Omron CX-Programmer project NewProject (CX-Programmer 9.61)

# PLC PLC_Pick: CP1H XA

## Global symbols (name address type ; comment)
0.00 BOOL  ; Start
0.01 BOOL  ; EmitBox
0.02 BOOL  ; EmitBox2
0.03 BOOL  ; Stop
0.04 BOOL  ; Dif1
0.05 BOOL  ; Dif2
0.06 BOOL  ; GrabDet
0.07 BOOL  ; Dif3
0.08 BOOL  ; Dif4
100.00 BOOL  ; M1
100.01 BOOL  ; M2
100.02 BOOL  ; M3
100.03 BOOL  ; M4
100.04 BOOL  ; M4
10.00 BOOL  ; Con6m
10.01 BOOL  ; Con2m1
10.02 BOOL  ; Con2m2
10.03 BOOL  ; BoxEmitter
10.04 BOOL  ; StoperRoll
10.05 BOOL  ; MZ
10.06 BOOL  ; MX
10.07 BOOL  ; Grab
10.08 BOOL  ; StoperBlade
T0000 BOOL  ; Timer1
T0001 BOOL  ; Timer2
T0002 BOOL  ; Timer3

## Program NewProgram1 (cyclic task 0)

### Section Section1

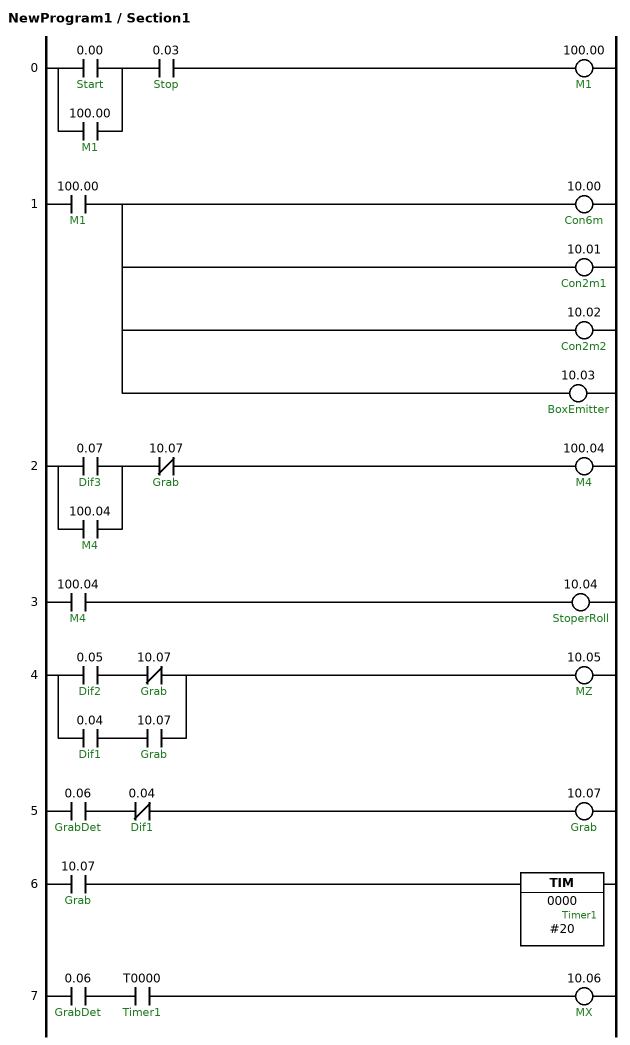
; rung 0
LD 0.00  ; Start
OR 100.00  ; M1
AND 0.03  ; Stop
OUT 100.00  ; M1
; rung 1
LD 100.00  ; M1
OUT 10.00  ; Con6m
OUT 10.01  ; Con2m1
OUT 10.02  ; Con2m2
OUT 10.03  ; BoxEmitter
; rung 2
LD 0.07  ; Dif3
OR 100.04  ; M4
ANDNOT 10.07  ; Grab
OUT 100.04  ; M4
; rung 3
LD 100.04  ; M4
OUT 10.04  ; StoperRoll
; rung 4
LD 0.05  ; Dif2
ANDNOT 10.07  ; Grab
LD 0.04  ; Dif1
AND 10.07  ; Grab
ORLD
OUT 10.05  ; MZ
; rung 5
LD 0.06  ; GrabDet
ANDNOT 0.04  ; Dif1
OUT 10.07  ; Grab
; rung 6
LD 10.07  ; Grab
TIM 0000 #20  ; Timer1
; rung 7
LD 0.06  ; GrabDet
AND T0000  ; Timer1
OUT 10.06  ; MX

### Section END
; rung 0
END(001)